FUNCTION_BLOCK FB_TestA IMPLEMENTS ITF_MyTest
VAR_INPUT
END_VAR
VAR_OUTPUT
END_VAR
VAR
	b1: BOOL;
	r32: REAL;
	str : STRING;
END_VAR

{warning 'Agregar implementación de método'}
METHOD METH1 : BOOL
METH1 := TRUE;
END_METHOD

{warning 'Agregar implementación de método'}
METHOD METH2 : STRING
METH2 := 'FB_TestA';
END_METHOD

{warning 'Agregar implementación de método'}
METHOD METH3 : REAL
METH3 := 3.14;
END_METHOD

{warning 'Agregar implementación de propiedad'}
PROPERTY Prop1 : BOOL
GET
Prop1:= b1;
END_GET
SET
b1 := Prop1;
END_SET
END_PROPERTY

{warning 'Agregar implementación de propiedad'}
PROPERTY Prop2 : REAL
GET
Prop2 := r32;
END_GET
SET
r32 := Prop2;
END_SET
END_PROPERTY

{warning 'Agregar implementación de propiedad'}
PROPERTY Prop3 : STRING
GET
Prop3 := str;
END_GET
SET
str := Prop3;
END_SET
END_PROPERTY

END_FUNCTION_BLOCK

(* stored: Version 1.1.0.1, ProductVersion 3.1.4024.12
   POU FB_TestA: Id {5a20f7d0-cac5-4a46-a04f-5f725d6bf91a}, SpecialFunc None
   Method METH1: Id {f9667a7b-55fd-4805-afa2-998d7cb2ba3b}
   Method METH2: Id {619e2910-40fc-4cba-a6fb-0b11e0aaad6a}
   Method METH3: Id {bca9ada1-a130-4cb4-a472-84c69b50f3b9}
   Property Prop1: Id {1cf77579-683c-4d7c-a6a2-6d797d8ef047}
   Get Get: Id {2d387ef6-99ef-4da2-9575-0955367d3e48}
   Set Set: Id {55a32bd6-0d32-4f52-ac97-774d2af1ee6b}
   Property Prop2: Id {d1fa0ce0-ffd1-48b4-a230-9c92aa2c9214}
   Get Get: Id {11bdbaed-576e-4945-821e-17de4d43a382}
   Set Set: Id {2152ab76-281a-4060-91f8-a204c1674ceb}
   Property Prop3: Id {d581feda-d2aa-4623-8abc-edfc5e50ff93}
   Get Get: Id {fb96d624-800e-4d04-9104-32f220c3a7a6}
   Set Set: Id {2377af72-a137-4f95-add6-bc1241087ca1} *)
